{attribute 'GeneratedUsingTerminal: ELX3351-0000-0016'}
{attribute addProperty BoxType "ELX3351-0000-0016"}
{attribute addProperty Id "StatusAT %I*Status_D17852406"}
{attribute addProperty CRC "4000008628"}
{attribute addProperty Size "6"}
TYPE RMB_Status_EE6B49B4 EXTENDS InputBase_8311D824 :
STRUCT
	{attribute addProperty Name "Status"}
	Status AT %I* : Status_D1785240;
END_STRUCT
END_TYPE

(* stored: Version 1.2.0.0, ProductVersion 3.1.4024.9
   DUT RMB_Status_EE6B49B4: Id {0a0ce0af-37d9-4613-a79e-d5ed7021f535} *)
